{attribute 'GeneratedUsingTerminal: EL3423-0000-0016'}
{attribute addProperty BoxType "EL3423-0000-0016"}
{attribute addProperty Id "Reactive_EnergyAT %I*LINT8Reactive_Positive_EnergyAT %I*ULINT8Reactive_Negative_EnergyAT %I*ULINT8"}
{attribute addProperty CRC "4009877245"}
{attribute addProperty Size "24"}
TYPE Total_Reactive_EF01DEFD EXTENDS InputBase_8311D824 :
STRUCT
	{attribute addProperty Name "Reactive_Energy"}
	Reactive_Energy AT %I* : LINT;
	{attribute addProperty Name "Reactive_Positive_Energy"}
	Reactive_Positive_Energy AT %I* : ULINT;
	{attribute addProperty Name "Reactive_Negative_Energy"}
	Reactive_Negative_Energy AT %I* : ULINT;
END_STRUCT
END_TYPE

(* stored: Version 1.2.0.0, ProductVersion 3.1.4024.9
   DUT Total_Reactive_EF01DEFD: Id {5761d88f-21ff-4d55-b761-76d4b91890ed} *)
